{attribute 'GeneratedUsingTerminal: EK1100-0000-0018'}
{attribute addProperty BoxType "EK1100-0000-0018"}
{attribute addProperty Id "Beckhoff_ER2xxxEK1122Beckhoff_ER2xxxEK1122_73471FC4910"}
{attribute addProperty CRC "3470310182"}
{attribute addProperty Size "910"}
TYPE Beckhoff_ER2xxx_CED8BB26 EXTENDS EK1100_1FC0878B :
STRUCT
	{attribute addProperty Name "Beckhoff_ER2xxxEK1122"}
	Beckhoff_ER2xxxEK1122 : Beckhoff_ER2xxxEK1122_73471FC4;
END_STRUCT
END_TYPE

(* stored: Version 1.2.0.0, ProductVersion 3.1.4024.9
   DUT Beckhoff_ER2xxx_CED8BB26: Id {0b1c802e-6f4b-411b-bbde-1a61dca6b68d} *)
